(*Instances*)
	HMI:HMI_TemplateMachinePart;						//All HMI related variables
	Tmr_Empty:TON;										//Timer detection machine is empty*)
	Tmr_Initialisation:TON;								//Timer template*)
	Tmr_TestServoVelo:ton;
	Tmr_Wrn_NoSupply:ton;
	//Signal		>> outputs high / low. It can be used for any signal (that is not a sensor).
	SN_DscReadyToReceive:cntrl_InputHmiSts;					//Signal discharge ready to receive products
	//PB_Safe 		>> HMI safe button. This block automatically outputs low signal if the HMI loses connection for more than x-time
	PBsf_Example:utl_PB_HmiSafe;						//Safe pushbutton
	
	(*EXAMPLE how to init setpoint variables (normally you are not allowed to write these!) OR any variable of an instance
		use f2 >> select you setpoint type, for this I've chosen HMI_SP_Sensor >> insert with arguments >> this wil show up:
			HMI_SP_Sensor := (
				TMR_Muting:= , 
				TMR_DelayDetected:= , 
				TMR_DelayUndetected:= , 
				TMR_DelayErrorDetect:= , 
				TMR_DelayErrorUndetect:= );
		with this info you can init the setpoints of the cntrl_Sensor block like this:*)				
	
	//cntrl_Sensor	>> outputs: product detected / not detected. It can be used for any detection for example: airpressure, an object, etc.	
	//* If you init setpoints like this, then these values will only be used at first time download of the block. 
	// >> you will have to do a "plc" / "reset origin"
	PC_ProductInfeed:cntrl_Sensor(
		//fb_init
		Options:= eSensorConfig.InputNO)
		//Example how to preset setpoint variables
		:=(
			HMI:=(
				SP:=(
					TMR_DelayDetected:=T#100MS , 
					TMR_DelayUndetected:= T#101MS, 
					TMR_DelayErrorDetect:= T#2S1MS, 
					TMR_DelayErrorUndetect:= T#2S2MS)));	//Photocell product infeed position
	
	
	PC_PlanoBufferLL: cntrl_Sensor(
		Options:= eSensorConfig.Default);					//Photocell planobuffer low level 	
					
 
	//Valve			>> used to control cylinders with valves and reedcontacts
	Cyl_Example:cntrl_Valve
		(Options:= eValveConfig.Default);	

	//Motor			>> standard motor with forward/reverse + ana speed all direct IO
	Mtr_Example:cntrl_Motor(
		Options:= eMotorConfig.Default, 
		TmrDirectionChange:= T#500MS, 
		MinAllowedSpeed:= 25, 
		DAC_0PrctValue:= 0, 
		DAC_100PrctValue:= 0);
	
	//FreqDrive	ControlTechniques C300	>> Frequency drive motor, this one is controlled by ethercat
	Fdr_CtExample:cntrl_FDR_ControlTech(
		Options:= eFdrGeneric_Config.WithMaintSwitch, 
		UnitsToOutputFactor:= 30);

	//FreqDrive	Lenze I550 >> Frequency drive motor, this one is controlled by ethercat
	Fdr_LzExample:cntrl_FDR_Lenze(
		Options:= eFdrGeneric_Config.WithMaintSwitch, 
		UnitsToOutputFactor:= 30);

	//The interrol roller-drive BI can be used as frequency drive but also as a Cia402 positioning device >> for test configged as positioning device
	Srv_Interrol: cntrl_FDR_Interrol(
		Options:= eFdrGeneric_Config.ExternalRunStates, //this tells the base block to hand over control to the child block for the running-states 
		UnitsToOutputFactor:= 1);

	//Servo			>> Beckhoff servo drive
	Srv_Example:cntrl_Servo(
		TMR_PowerSave:=T#30S,			//time before entering powersave mode 0=disabled (if no command is given then power down after this time @ any command is reset timer) !It takes some time to awake the servo
		EnableSoftLimits:=FALSE,		//enable software limits (with button manual disable hw-limits, the parameter in the nc-task is set to 0, we need to know if it should be reenabled afterwards
		InputNrHomingSensor:=-1,			//input nr for the sensor in "axis_ref_Extended.I_DigitalInputs" -1 == disabled
		InputNrHwLimitNeg:=-1,			//input nr for the sensor in "axis_ref_Extended.I_DigitalInputs" -1 == disabled
		InputNrHwLimitPos:=4,			//input nr for the sensor in "axis_ref_Extended.I_DigitalInputs" -1 == disabled
		JogMinusOffHomeSensor:=FALSE,	//"jog-"  when moving off homing sensor (if false then jog+ is used) in homing function
		HomingsensorIs_NC:=FALSE,		//the homing sensor is of type normally closed (note limitswitches are always normally closed)
		TmrErr_JogOffHomeSensor:=T#3S,	//time to try and jog off homing sensor t#0S = disable
	
		HomeTorqueSpeed:=0,						//Speed to use for homing in torque mode
		HomingMode:= eSrvHomingModes.Direct,	//homing mode to use >> Default, Direct, Set, Reset, TorquePositiveDirection, TorqueNegativeDirection
		CouplingSyncPosFirst:=FALSE,			//at couple command, sync the position first to the master axis
		SPD_CouplingSyncSpeed:=0,				//speed to use when syncing position for coupling
		DST_CouplingSyncMaxDiff:=0,				//max difference allowed when sync couling >> otherwise error
		//MAKE SURE VALUE IS CORRECT (set to 0 to use nc-task configured dynamics)
		DEC_EmergencyError:=5000,				//deceleration ramp to use for emergency/error situation <= 0 means use default ramp
		//SET LOWER!!! >> jog=50, velo=250
		SPD_JOG_Max:=5000,						//max allowed allowed jog speed (also used to jog of homing sensor during homing)
		SPD_AbsModVel_MaxMan:=5000				//max allowed speed in manual absolute,velocity, modulo mode	
		);
	//Ganty			>> Gantry controlled with 2 beckhoff servo's connected to the same drive-belt
	Gantry_Example:cntrl_SingleBeltGantry(
			IsHomingUp:= TRUE, 
			IsHomingRight:= TRUE, 
			TMR_DelayPowerSave:= T#1M , 
			SPD_MaxJog:= 50, 
			SPD_MaxMove:= 150);
	
	//Robot			>>customized library robot block
	Rbt_Unloading: cntrl_RbtFanucUnloadingRobot();
			
	//VacuumGenerator	>>	Vacuumgenerator with blowoff controlled by IO
	Vcg_Suckers : cntrl_VacuumGenerator(
		//fb_init
		Options:= eVacuumGeneratorConfig.Default + eVacuumGeneratorConfig.DropVacAtVacErr)
		//interal vars
		:=(PS_VacuumOk:=(
			HMI:=(
				SP:=(
					TMR_DelayErrorDetect := T#2S,
					TMR_DelayErrorUnDetect := T#2S))));

	//Omron FH			>> Omron camera's controlled by an omron FH-controller over ethercat
	Cam_OmronFh: Cntrl_OmronFh;
	//Omron FH controlled by ethernet
	Cam_OmronFhEth: cntrl_OmronFhEth;
	Cam_OmronFhEthResult: utl_OmronFhEthResult_Template;
	Cam_OmronFhEthSimMessage:STRING := '1;65.9;85.4;-78.3;75;1;$R';

	//Omron smartcam	>> Omron smart camera's over ethernet / direct IO for trigger
	Cam_OmronSmartCam: Cntrl_OmronMicroScan(
		AlwaysConnected:= FALSE, 	//try to connect to camera even if no auto_k 
		JobNr:= 1, 					//default job nr to load if job load command is given (can be changed with property)
		UseIoTrigger:= FALSE);		//instead of trigger over ethernet, send trigger by real output
	

(*Inputs / Outputs*)
	//note> since there is a logged library input-block (cntrl_InputXXX) 
END_VAR

(*
	Update HMI variables
	Check if an error is active >> set Q_ProgStatus.Prog_Errror
*)
	HMI.M_Update(	I_OrgControl:= I_Organiser, 	//used for reset manuals/errors commands
					I_HMI_Parent := 0, 				//This is top level, no error propagation
					I_ERR:= HMI.ERR,				//The update function will check for error changes (signal to the hmi to update errors) + reset errors
					I_WRN:= HMI.WRN,				//The update function will check for warning changes (signal to the hmi to update errors)
					I_MAN:= HMI.MAN);				//The update function will reset manuals @ organiser request
			
(*	Simulation*)
	//if simulation active >> ..
	IF(Glbl.Sim_MyMachinePart) THEN A_Simulation();END_IF

(*	Exceptions & step-controller*)
	A_Exceptions();
		
(*	Step transitions*)
	//if not in exception >> execute step transitions
	IF (	NOT HM_ProgStatus.Prog_Exception)
	THEN 
		A_StepTransitions();
	END_IF
	
(*	Activations*)
	//Reset all outputs controlled by states
	A_ActivationsInit();
	//Activate outputs controlled by state
	A_ActivationsState();
	//Activate outputs not controlled by state + call all instances
	A_ActivationsAlways();
	
(*update organiser with scam status*)
	A_UpdateOrganiserProgstatus();

ACTION A_ActivationsAlways:
(*
	State undependant activations + instance calls
*)
//Internal flags
	//if running and product detected or supply might be supplying products > reset empty status
	IF (	I_Organiser.EnableDevices_K
			AND (	PC_ProductInfeed.Q_DetectedDebounced
					OR NOT I_STS_SUP_Empty))
	THEN
		HM_Empty := FALSE;
	END_IF

//Warnings/Statusses
	Q_STS_Empty := HM_Empty;
	HMI.STS.IsEmpty := HM_Empty; //can be used to indicate on the HMI this machinepart is empty
	Q_STS_RefillPlanos := NOT PC_PlanoBufferLL.Q_DetectedDebounced;
	HMI.WRN.PlanoBufferNeedsRefill := NOT PC_PlanoBufferLL.Q_DetectedDebounced;
	HMI.WRN.NotRdyRcv_Discharge := 	I_Organiser.EnableDevices_K
									AND NOT SN_DscReadyToReceive.Q;

	//if pulse 1s >> increase hmi test int until max reached which resets to 0
	IF(BknGlbl.Blink_P_1s)
	THEN
		HMI.STS.testInt := HMI.STS.testInt + 1; IF(HMI.STS.testInt > 5) THEN HMI.STS.testInt := 0; END_IF;
	END_IF

//Timers
	Tmr_Empty(	//IN:= ,
				PT:= T#30S );	
	
	Tmr_Initialisation(
		//IN:= ,
		PT:= T#3S);
		
	Tmr_TestServoVelo(	//IN:= , 
						PT:= T#5S);

//Instance calls
	//Safe button (protection against loss of communication with the HMI >> will set state to low)
	PBsf_Example();

	PC_ProductInfeed(
		I_HMI_Parent:= HMI,
		I_K_SimulationActive:= Glbl.Sim_MyMachinePart, 
		I_OrgControl := I_Organiser);
		//I_SimulateState:= ,
		//I_K_ErrNotState:= ,
	
	//Logged counter: example how we can count the debounced falling edges of a photocell
		IF(PC_ProductInfeed.Q_DetectedDebounced_RE) THEN 	PC_Example_Count.V := PC_Example_Count.V + 1; END_IF
	
	PC_PlanoBufferLL(
		I_HMI_Parent:= HMI,
		I_OrgControl:= I_Organiser,
		I_K_SimulationActive:= Glbl.Sim_MyMachinePart,
		I_SimulateState:= eSensorState.Detected, 
		I_ErrNotState:= eSensorState.None);
	
	SN_DscReadyToReceive(
		I_K_SimulationActive:= Glbl.Sim_MyMachinePart, 
		//I_K_SimulateOn:= 
		);
	
	Cyl_Example(
		I_HMI_Parent:= HMI,
		I_K_SimulationActive:= Glbl.Sim_MyMachinePart, 
		I_ES_OK:= I_K_ES_OK, 
		I_OrgControl:= I_Organiser,  
		//I_K_AutoIn:=,
		//I_K_AutoOut:=,
		);
		
	Vcg_Suckers(
		I_HMI_Parent:= HMI,
		I_K_SimulationActive:= Glbl.Sim_MyMachinePart,
		I_ES_OK:= I_K_ES_OK, 
		I_OrgControl:= I_Organiser, 
		//I_K_Auto_Vacuum:= , 
		//I_K_Auto_BlowOff:= , 
		);

	Mtr_Example(
		I_HMI_Parent:= HMI,
		I_K_SimulationActive:= Glbl.Sim_MyMachinePart, 
		I_ES_OK:= I_K_ES_OK, 
		I_OrgControl:= I_Organiser, 
		//I_K_Auto_Fwd:= , 
		//I_K_Auto_Rev:= , 
		I_Spd_AutoPrct:= -1, //>>use IO_SP.Spd_Default instead
	);
		
	Fdr_CtExample(
		I_HMI_Parent:= HMI,		
		I_K_SimulationActive:= Glbl.Sim_MyMachinePart, 
		I_ES_OK:= I_K_ES_OK, 
		I_OrgControl:= I_Organiser,  
		//I_K_Auto_Fwd:= ,
		//I_K_Auto_Rev:= , 
		//I_SPD_AutoPrct:= , 
		);
		
	Fdr_LzExample(
		I_HMI_Parent:= HMI, 
		I_K_SimulationActive:= Glbl.Sim_MyMachinePart, 
		I_ES_OK:= I_K_ES_OK, 
		I_OrgControl:= I_Organiser, 
		//I_K_RunFwd:= , 
		//I_K_RunRev:= , 
		//I_Speed:= 
		);
	
	
	//todo debug test
	Srv_Example.I_K_PosAbsolute R= HM_DebugServoRestart;
	Srv_Example(
		I_HMI_Parent:= HMI,
		I_PTR_MasterAxis:=0, 
		I_K_SimulationActive:= Glbl.Sim_MyMachinePart, 
		I_ES_OK:= I_K_ES_OK, 
		I_OrgControl:= I_Organiser, 
		//..several commands.. 
		I_CPF_CoupleFactor:= 1, 
		I_K_CoupleAxis:= FALSE, 
		I_K_UnCoupleAxis:= FALSE, 
		I_K_ExternalSetpoint:= FALSE); HM_DebugServoRestart := FALSE;
		
		(*log actual position / velocity. 
			*Constantly logging positions causes a lot of data for the logger!
			This is why in the servo block no position logging is done and you have to add it manually if you need it.
				>>decrease logging data volume by setting trigInterval and trigDeviation and add an elogGroup which is only activated when you need it
				>>Or only log at step transition
					IF(myStepCondition)
					THEN
						SRV_ExamplePos.V := TO_REAL(fbSrv_Example.P_STS_ActPosition);
						//>
						eMyStep:= blablabla;
					END_IF
		Done as below causes a lot of data
		*)
		Srv_Example_Velo.V := TO_REAL(Srv_Example.P_STS_ActVelocity); 
		
		(*Very specific example where the configuration is changed based on certain conditions>> for this example normally the man-speeds are only set in fb_init()*)
		//if in manual mode
		IF(I_Organiser.Manual_K AND FALSE)
		THEN
			//if servo is NOT coupled >> limit to lower value for safety
			IF(NOT Srv_Example.P_STS_IsCoupled) 
			THEN 
				Srv_Example.P_CFG_SPD_ABSMODVEL_MaxMan := 5;
				Srv_Example.P_CFG_SPD_JOG_MaxMan := 5;
			ELSE
				Srv_Example.P_CFG_SPD_ABSMODVEL_MaxMan := 500;
				Srv_Example.P_CFG_SPD_JOG_MaxMan := 100;
			END_IF
		END_IF
		
	Srv_Interrol(
		I_HMI_Parent:= HMI, 
		I_OrgControl:= I_Organiser, 
		I_K_SimulationActive:= Glbl.Sim_MyMachinePart, 
		I_ES_OK:= I_K_ES_OK, 
		I_K_Auto_Fwd:= FALSE, 		//not used in this example (can be used!) 
		I_K_Auto_Rev:= FALSE, 
		I_Speed:= -1,				// <0 = block will use internal setpoint value 
		//I_K_AbsPositioning:= , 	//only used command in this example
		//I_Position:= , 
		);
	
	Gantry_Example(
		I_HMI_Parent:= HMI,
		I_K_SimulationActive:= Glbl.Sim_MyMachinePart,
		I_ES_OK:= I_K_ES_OK, 
		I_OrgControl:= I_Organiser,
		//I_Auto_K_Homing:= , 
		//I_Auto_K_MoveToPos:= , 
		//I_Auto_POS_MoveToPos:= , 
		//I_Auto_SPD_MoveToPos:= 
	);
	
	Rbt_Unloading(
		I_HMI_Parent:= HMI, 
		I_OrgControl:= I_Organiser, 
		I_K_SimulationActive:= Glbl.Sim_MyMachinePart, 
		I_ES_OK:= I_K_ES_OK, 
		I_K_ProgramSelect:= , 
		I_SP_ProgramNr:= , 
		Q_K_ProgramSelect_OK=> );
	
	Cam_OmronSmartCam(
		I_HMI_Parent:= HMI,
		I_K_SimulationActive:= Glbl.Sim_MyMachinePart,
		I_OrgControl:= I_Organiser, 
		//I_K_Trigger:= , 
		//I_K_AutoCal:= , 
		//I_K_QuickFocus:= , 
		//I_K_LoadJob:= , 
		IO_DataReceive:= HM_CamReceivedData, 
		);
		//just for debugging, should be removed
		//data should normally be handled at the state transition when waiting for trigger ok
		IF(Cam_OmronSmartCam.Q_K_Trigger_Ok)
		THEN
			//note: this boikon library block will take care not to overflow the destination memory
			utl_Any_CopyWithOffset(
				I_Destination:= HMI.STS.OmronSmartCamLastResult, 
				I_Source:= HM_CamReceivedData, 
				I_WriteOffset:= 0);
		END_IF
		
	Cam_OmronFh(
		I_HMI_Parent:= HMI,
		I_K_SimulationActive:= Glbl.Sim_MyMachinePart,
		I_OrgControl:= I_Organiser,
		//I_K_Trigger:= , 
		//I_K_TriggerNextResult:= , 
		//I_K_ChangeGroup:= , 
		//I_K_LoadScene:= , 
		//I_SceneToLoad:= , 
		);
	
	(*Simple example of handling data received by controller. 
	I recommend doing this in the step transition and directly connect it to the desired location and using return value of the function instead of doing it here
	the disadvantage of doing it like this that everything inside the block is executed continiously and hogs the processor.
	Recommended way @ step transitions: 
		IF(utl_OmronCameraResult(..,..,myBuffer)) 
		THEN 
			//>>
			eS:=xxx.CamResultOK;
		ELSE
			//>>
			eS:= xxx.CamResultNOK;
		..
	*) 

	Cam_OmronFhEth(
		I_HMI_Parent:= HMI, 
		I_K_SimulationActive:= Glbl.Sim_MyMachinePart,
		I_SimulationTrigResult:= Cam_OmronFhEthSimMessage,
		I_OrgControl:= I_Organiser, 
		I_ReceiveBuffer:= HM_CamOmronFhEthReceivedData, 
		I_K_LoadScene:= ,
		I_K_UpdateStatus:= , 
		//I_K_Trigger:= 
			);
			
		//block that will resolve results from camera measurement output
		Cam_OmronFhEthResult(
			I_K_TrigOk:= Cam_OmronFhEth.Q_K_TriggerOk,
			I_DataUsedSize:= Cam_OmronFhEth.Q_STS_TriggerNrBytesReceived, 
			I_Data:= HM_CamOmronFhEthReceivedData);
END_ACTION

ACTION A_ActivationsInit:
(*	
	Initialisation of state dependant activations
*)
HM_ProgStatus.Prog_Rest := FALSE;
Q_SN_SUP_Request := FALSE;
PC_ProductInfeed.I_ErrNotState := eSensorState.None;
Mtr_Example.I_K_Auto_Fwd := FALSE;
Mtr_Example.I_K_Auto_Rev := FALSE;
Fdr_CtExample.I_K_Auto_Fwd := FALSE;
Fdr_CtExample.I_K_Auto_Rev := FALSE;
Fdr_LzExample.I_K_Auto_Fwd := FALSE;
Fdr_LzExample.I_K_Auto_Rev := FALSE;
Cyl_Example.I_K_AutoIn := FALSE; 
Cyl_Example.I_K_AutoOut := FALSE;
Vcg_Suckers.I_K_Auto_BlowOff :=FALSE;
Vcg_Suckers.I_K_Auto_Vacuum :=FALSE;
Srv_Example.I_K_Homing:= FALSE;
Srv_Example.I_K_PosAbsolute:= FALSE;
Srv_Example.I_K_Velocity := FALSE;
Srv_Interrol.I_K_AbsPositioning := FALSE;
Cam_OmronFh.I_K_Trigger := FALSE;
Cam_OmronFh.I_K_TriggerNextResult := FALSE;
Cam_OmronFh.I_K_ChangeGroup:= FALSE;
Cam_OmronFh.I_K_LoadScene:= FALSE;
Cam_OmronFhEth.I_K_Trigger:= FALSE;
Cam_OmronSmartCam.I_K_AutoCal := FALSE;
Cam_OmronSmartCam.I_K_LoadJob := FALSE;
Cam_OmronSmartCam.I_K_QuickFocus := FALSE;
Cam_OmronSmartCam.I_K_Trigger := FALSE;
Rbt_Unloading.I_K_DropBasket := FALSE;


Tmr_Empty.IN := FALSE;
Tmr_TestServoVelo.IN := FALSE;
Tmr_Initialisation.IN := FALSE;
Tmr_Wrn_NoSupply.IN := FALSE;

HM_DebugMultiStep_ResetInActivations := false;
END_ACTION

ACTION A_ActivationsState:
(*
	State dependant activations
*)
CASE State.eS OF
	eTMP.TotalReset:
		;
	
	eTMP.InitCyl:
		Cyl_Example.I_K_AutoIn:= TRUE; 
	
		(*Warnings/Errors*)
			//a sensor error can be triggered by activating the I_K_ErrNot.... input >> uses internally a timer
			//usually we want the machine to be empty in the init phase so setting error here if it is not
			PC_ProductInfeed.I_ErrNotState := eSensorState.Undetected; 
			//or an error can also be set directly
			//IF( [some condition] ) then IO_ERR.PC_ProductPassedStopper.NotLow := true; END_IF  !!!Errors must be a set! 
	
	eTMP.InitSrv:
		Cyl_Example.I_K_AutoIn:= TRUE; 
		Mtr_Example.I_K_Auto_Fwd:= TRUE;
		Srv_Example.I_K_Homing:= TRUE;
		Tmr_Initialisation.IN:= Mtr_Example.P_STS_Running;
	
		(*Warnings/Errors*)
			//S= >> SET!!! , all errors have to be set. In tc3 we can now use S= instead of "IF(..)THEN err:=true; end_if"
			HMI.ERR.InitNotEmpty S= PC_ProductInfeed.Q_DetectedDebounced;  	//detection machine is not empty during init
			PC_ProductInfeed.I_ErrNotState := eSensorState.Undetected;			//it is nice to also trigger this error, especially if there are multiple sensors. This at a faulty sensor the operator knows which sensor causes the problem
	
	eTMP.InitCamQuickFocus:
		Cyl_Example.I_K_AutoIn:= TRUE; 
		Cam_OmronSmartCam.I_K_QuickFocus:= TRUE;
	
	eTMP.InitCamLoadJob:
		Cyl_Example.I_K_AutoIn:= TRUE; 
		Cam_OmronFh.I_K_LoadScene:= TRUE;
		Cam_OmronFh.I_SceneToLoad:= 2;
		Cam_OmronSmartCam.I_K_LoadJob:= TRUE;
		Cam_OmronSmartCam.P_SP_JobToLoad:= 1; //note: these kind of variables can also be set @RE step (>>when stepping from previous step to here)			(*Internals*)
			
	eTMP.Rest:
		HM_ProgStatus.Prog_Rest:= TRUE;
		Q_SN_SUP_Request:= TRUE;
		Cyl_Example.I_K_AutoIn:= TRUE; 
		
		(*Warnings/Errors*)
			//just an example, no need to add this specific warning. The camera itself generates an error if it fails to connect
			HMI.WRN.CameraNotReady:= 	I_Organiser.EnableDevices_K
										AND NOT Cam_OmronSmartCam.Q_STS_Ready;  
			
			//if the supply is running >> the photocell should get high after x-time, set error detection of the pc
			IF(	I_SN_SUP_Request_OK
				AND NOT I_STS_SUP_Empty
				AND I_Organiser.EnableDevices_K)
			THEN
				PC_ProductInfeed.I_ErrNotState:= eSensorState.Detected; 
			END_IF

	eTMP.SrvPosStart:
		Cyl_Example.I_K_AutoIn:= TRUE; 
		Srv_Example.I_K_PosAbsolute:= TRUE;
		//there are multiple ways of setting a speed, this way per step the speed can be changed but it can also set fixed at the servo block
		//also note how for the gripper, settings are applied at the step change >>better way if during the step the settings do not have to change
		Srv_Example.I_SP_Speed:= 50;
		Srv_Interrol.I_K_AbsPositioning := TRUE; 
		
	eTMP.SrvPosStartInterl:
		Cyl_Example.I_K_AutoIn:= TRUE;
		Rbt_Unloading.I_K_DropBasket := true;
		
		(*Warnings/Errors*)
			PC_ProductInfeed.I_ErrNotState:= eSensorState.UnDetected; 

	eTMP.SrvPosEnd:
		Cyl_Example.I_K_AutoIn:= TRUE;
		Srv_Example.I_K_PosAbsolute:= TRUE;
		Srv_Example.I_SP_Speed:= 50; //there are multiple ways of setting a speed, this way per step the speed can be changed but it can also set fixed at the servo block
		Srv_Interrol.I_K_AbsPositioning := TRUE;
		
	eTMP.SrvPosEndIntrl:
		Cyl_Example.I_K_AutoIn:= TRUE;
		
	eTMP.CylOut:
		Cyl_Example.I_K_AutoOut:= TRUE;
		Vcg_Suckers.I_K_Auto_Vacuum:=TRUE;
		
	eTMP.CylIn:
		Cyl_Example.I_K_AutoIn:= TRUE;
		Vcg_Suckers.I_K_Auto_BlowOff:=TRUE;	
		
	eTMP.MtrStartFwd:
		Cyl_Example.I_K_AutoIn:= TRUE;	
		Mtr_Example.I_K_Auto_Fwd:= TRUE;

		//fdr's speed = block input
		Fdr_CtExample.I_K_Auto_Fwd:= TRUE;
		Fdr_CtExample.I_Speed:= -1; //<0 means use HMI.SP.Speed
		Fdr_LzExample.I_K_Auto_Fwd:= TRUE;
		Fdr_LzExample.I_Speed := 50;
		
	eTMP.MtrStop:
		Cyl_Example.I_K_AutoIn:= TRUE;
	
	eTMP.MtrStartRev:
		Cyl_Example.I_K_AutoIn:= TRUE;	
		Mtr_Example.I_K_Auto_Rev:= TRUE;

		//fdr's speed = HMI.SP
		Fdr_CtExample.I_K_Auto_Rev:= TRUE;
		Fdr_CtExample.I_Speed:= 75; //<0 means use HMI.SP.Speed
		Fdr_LzExample.I_K_Auto_Rev:= TRUE;
		Fdr_LzExample.I_Speed := -1; //<0 means use HMI.SP.Speed

	eTMP.CamReady:
		Cyl_Example.I_K_AutoIn:= TRUE;			
	
	eTMP.CamTrig:
		Cyl_Example.I_K_AutoIn:= TRUE;
		Cam_OmronFh.I_K_Trigger:= TRUE;
		Cam_OmronFhEth.I_K_Trigger:= TRUE;
		Cam_OmronSmartCam.I_K_Trigger:= TRUE;	
		
(*
	S_Example:
		//Comm signals
		//Timers
		//Internals
		//Controls
		//Warnings
		//Errors
*)

END_CASE
END_ACTION

ACTION A_Exceptions:
(* State transition controller
	Handles multistep + step hold + statusses for hmi + logging*) 
		//>>must be before all method calls, since the input arguments are used
	State(I_OrgControl := I_Organiser);

(*Exceptions
	Here exeptions are handled.
	*most basic version:
		Rest U_0 := Q_ProgStatus.Prog_Exception:=false
			the main program is executed
	
		Rest >> Error := Q_ProgStatus.Prog_Exception:=true
		1)	@ any error >> exception state (U1_0)
			this will freeze the main program states
		2)	if the organiser is back in an automatic state and there are no errors
			it will step to U1_2 and from there to the idle state U_0
			*TODO TEMPLATE >> if needed, do actions on this transition (rarely used)
				But you could for example at a specific error force the main program to a recovery step
			
			
		Rest >> Totalreset := Q_ProgStatus.Prog_Exception:=true
		1)	@ organiser total reset command >> exception total reset (U1_1)
		
		2)	@ NOT organiser total reset command >> 
				>> now bits that need to be reset @ total reset are reset
				TODO Template >> add bits which needs to be reset
				>> the main program is reset to the first step (usually named: TotalReset)
				>>back to rest (U_0)

	**this described the basic version which can be used in 99% of the cases,
	you can adapt it to your needs. 
*)

CASE eE OF
	//rest
	U_0:
		
		//if program in error >> to error state
		IF(	HM_ProgStatus.Prog_Error
			AND NOT I_Organiser.TotalReset_K)
		THEN
			//>>
			eE := U1_0;
		//else if total reset command >> to total reset state
		ELSIF(	I_Organiser.TotalReset_K)
		THEN
			//>>
			eE := U1_1;
		END_IF

	//error
	U1_0:
		//if total reset command >> to total reset state
		IF(	I_Organiser.TotalReset_K)
		THEN
			//>>
			eE := U1_1;
			
		//else if no error active and organiser back in an automatic state
		ELSIF(	NOT HM_ProgStatus.Prog_Error
				AND I_Organiser.EnableDevices_K)
		THEN
			//>>
			eE := U1_2;
		END_IF

	//Total Reset
	U1_1:
 		//if total reset command dropped >> Reset program data and to unfreeze state
		IF(	NOT I_Organiser.TotalReset_K)
		THEN
			//Total reset main program
			State.M_Step(
				I_NewStep:= eTMP.TotalReset,
				I_StepCanBeHeld:= TRUE);
			
			//disable multistepping for 1 round
			{warning disable C0139}
			State.P_IsMultiStepRequired;

			//Reset main program flags
			HM_Empty:=FALSE;
			//only done as example/testing, should be removed
			HMI.ERR.ExampleAddPrioForHmiError := TRUE;
			
			//>>
			eE := U_0;
		END_IF
		
	//Unfreeze
	U1_2:
		//>>
		eE := U_0;

	ELSE
		eE := U_0;
END_CASE

//Detection program in exception
HM_ProgStatus.Prog_Exception := (eE > U_0);
END_ACTION

ACTION A_Simulation:
(*
	Code that only needs to be executed if simulation is active (this action is only called if sim is active)

	Notes:	
	-Cntrl_Servo/motor/valve already simulate their state correctly themselves, cntrl_StateSensor must be told which state to simulate >> example below
		Of course you could also add timers / other conditions (servo pos?!) for states
	
	-you can use ( Tmr_StateTime.PT > T# xxx) to start simulating things after the state has been active for a certain time
*)

//Initialise activations, which are controlled by the simulation steps
SN_DscReadyToReceive.I_K_SimulateOn := FALSE;
PC_ProductInfeed.I_SimulateState := eSensorState.Undetected;

(*Step activations*)
CASE State.eS OF
	eTMP.TotalReset:
	;

	eTMP.InitCyl:
	;
	
	eTMP.InitSrv:
	;

	eTMP.Rest:
		PC_ProductInfeed.P_BypassErrDetectionTime := State.P_StepTime + T#100MS; 
		
		//If delay time elapsed >> simulate sensor + discharge request
		IF(State.P_StepTime > T#1S) 
		THEN
			SN_DscReadyToReceive.I_K_SimulateOn := TRUE; 
			PC_ProductInfeed.I_SimulateState := eSensorState.Detected;
		END_IF
		
	eTMP.SrvPosStart:
	;
		
	eTMP.SrvPosStartInterl:
	;
END_CASE	

//feedback request to input
I_SN_SUP_Request_OK := Q_SN_SUP_Request;
END_ACTION

ACTION A_StepTransitions:
(*In this section all state transitions are made

	-no activations are done here (do this in A_Activations)
	-The transition to a new step is the ideal location to do rising edge settings
		IF(myCondition) THEN
			HM_CNT_Example := HM_CNT_EXAMPLE + 1; //example to count something
			fbSrv_Example.I_POS_Auto_Absolute := myNewPosition + someCalculated offset; //example to calculate endpoint for a servo
			//Note: you could set the servo speed here as well, but then you can't change the speed anymore during the movement
				probably (dependant on your situation) better to do it in activations.
			//>>
			step to next step
		END_IF

*)

(*Main program steps*)

//if stepping not locked, by steplock mode >> can be toggled in HMI to lock certain steps for commissioning/debugging
IF( NOT State.Q_K_LockSteps)
THEN
//Repeat until conditions to step to next state are false OR looped already twice (normally programs don't loop multiple times!)
REPEAT 
	CASE State.eS OF
		eTMP.TotalReset:
			//if initialise command from the organiser >> start initialisation
			IF ( I_Organiser.Init_K)
			THEN
				//>>
				State.M_Step(
					I_NewStep:= eTMP.InitCyl,
					//Optional: argument to log extra info for this step transition
					I_NewStepLogInfo:= CONCAT('TotalReset:', SYSTEMTIME_TO_STRING(BknGlbl.LocalSystemTime)),
					//>>@ true & HMI-stepmode is activated, then the next state will be locked until you press the button release step on the HMI (used for debugging / commissioning
					//!Do not enable for states in which things are cooking: (heater enabled / motor running / etc) or at least consider carefully potential dangers.
					I_StepCanBeHeld:= TRUE,
					//Optional: >> the repeat around this CASE-statement will NOT execute, the next step will take at least 1 cycle == activations for that step are executed 	
					I_BlockMultiStep:=TRUE); 
			END_IF

		
		eTMP.InitCyl:
			//if cylinder initialised and no products in the machine >> InitSrv
			IF( Cyl_Example.Q_STS_In
				AND NOT PC_ProductInfeed.Q_DetectedDebounced) //note: >> set error detection in activations!
			THEN
				//>>
				State.M_Step(
					I_NewStep:= eTMP.InitSrv,
					I_StepCanBeHeld:= TRUE);
			END_IF
			
		eTMP.InitSrv:
			//if servos homed and minimal time elapsed >> next state
			IF( Srv_Example.Q_K_HomingOk
				AND Tmr_Initialisation.Q) 
			THEN
				//>>
				State.M_Step(
					I_NewStep:= eTMP.InitCamQuickFocus,
					I_StepCanBeHeld:= TRUE);
			END_IF
			
		eTMP.InitCamQuickFocus:
			//if camera ready / quickfocus done >>..
			IF(	Cam_OmronFh.Q_STS_Ready
				AND Cam_OmronSmartCam.Q_K_AutoOrQuickCal_Ok)
			THEN
				//>>
				State.M_Step(
					I_NewStep:= eTMP.InitCamLoadJob,
					I_StepCanBeHeld:= TRUE);
			END_IF
			
		eTMP.InitCamLoadJob:
			//if camera's loaded jobs >. ..
			IF(	Cam_OmronFh.Q_SN_LoadScene_OK
				AND Cam_OmronSmartCam.Q_K_LoadJob_Ok)
			THEN
				//>>
				State.M_Step(
					I_NewStep:= eTMP.Rest,
					I_StepCanBeHeld:= TRUE);
			END_IF

		eTMP.Rest: 
			//if in automatic mode and supply delivered product and interlockings ok
			//>>SrvPosStart
			IF( I_Organiser.Auto_K
				AND NOT HM_Empty					//machine is not empty (inclusive supply)
				AND I_SN_SUP_Request_OK				//supply delivered product
				AND SN_DscReadyToReceive.Q 			//discharge is requesting products
 				AND PC_ProductInfeed.Q_DetectedDebounced 	//expected the sensor to be high >> activate error monitoring in activations

				//interlocking >> check blocks returned to rest/ready state
				AND Cam_OmronFh.Q_STS_Ready
				AND Cam_OmronFhEth.Q_STS_Ready
				AND Cam_OmronSmartCam.Q_STS_Ready
				AND Cyl_Example.Q_STS_In
				AND NOT Vcg_Suckers.Q_K_BlowOffOK 	
				AND NOT Vcg_Suckers.Q_K_VacuumOK
				AND NOT Srv_Example.Q_K_PosAbsoluteOk
				AND NOT Srv_Interrol.Q_STS_TargetReached)
			THEN
				//setting positions on step change, you could also constantly write these positions constantly in activations
				Srv_Example.I_SP_Position:= HMI.SP.POS_SrvBegin;
				Srv_Interrol.I_Position:= HMI.SP.POS_SrvBegin;
				
				//example on how to avoid concat(concat(concat(concat......)))))
				//NOTE: it is not the most performant because of all the fancy c#-linq-like stuff but it is the simplest and faster than concat
				// 		really fast is using utl_Any_CopyWithOffset directly (the databuilder is a wrapper around that function)
				DataBuilder.
					//assign databuffer
					M_SetTarget(HM_InfoString).
					//add a string that is not a variable otherwise use: M_WithData(HM_MyStringVar)
					M_WithStringLiteral('Last cycle time:').
					M_WithStringLiteral(TO_STRING(TO_REAL(BknGlbl.SystemTimeInTicks - HM_LastTicksStateRest)/10000000)).
					M_WithStringLiteral('s Servos target pos:').
					M_WithStringLiteral(TO_STRING(HMI.SP.POS_SrvBegin)); 
					
				//>>
				State.M_Step(
					I_NewStep:= eTMP.SrvPosStart,
					//just an example what you can do (add state info for logging purposes), this argument is optional
					I_NewStepLogInfo:= HM_InfoString,
					I_StepCanBeHeld:= FALSE);
				
				HM_LastTicksStateRest := BknGlbl.SystemTimeInTicks;	
			//if in semi-automode and the operator choose a special action >> do requested action
			ELSIF( 	I_Organiser.SemiAuto_K
					AND TRUE) //insert HMI.STS.TB_RequestSpecialAction
			THEN
				
				//>>
				State.M_Step(
					I_NewStep:= eTMP.SemiAutoStart,
					I_StepCanBeHeld:= TRUE);
					
				HM_LastTicksStateRest := BknGlbl.SystemTimeInTicks;
			END_IF

		eTMP.SrvPosStart:
			//if servo's reached commanded position
			IF( Srv_Example.Q_K_PosAbsoluteOk
				AND Srv_Interrol.Q_STS_TargetReached
				//interl. make sure not still high from previous action
				AND NOT Rbt_Unloading.Q_K_DropBasket_OK)
			THEN
				//>>
				State.M_Step(
					I_NewStep:= eTMP.SrvPosStartInterl,
					I_StepCanBeHeld:= TRUE); //enabling step lock, so we can see at the machine how the servo is positioned if done 
			END_IF
		
		eTMP.SrvPosStartInterl:
			//if robot done and interlockings with servo/supply done
			//>>SrvPosEnd
			IF( 	Rbt_Unloading.Q_K_DropBasket_OK
					AND NOT PC_ProductInfeed.Q_DetectedDebounced			//let's also check the sensor dropped again >> make sure to trigger error detection in activations
					AND NOT I_SN_SUP_Request_OK					//product was handled, check if supply acknowledges
					//interl. next step a command is given so we need to interlock here
					AND NOT Srv_Example.Q_K_PosAbsoluteOk
					AND NOT Srv_Interrol.Q_STS_TargetReached)		
			THEN
				//again setting position on step change, you could also constantly write these positions constantly in activations
				Srv_Example.I_SP_Position := HMI.SP.POS_SrvEnd;
				Srv_Interrol.I_Position:= HMI.SP.POS_SrvEnd;
				
				//>>
				State.M_Step(
					I_NewStep:= eTMP.SrvPosEnd,
					I_StepCanBeHeld:= FALSE);
			END_IF
			
		eTMP.SrvPosEnd:
			//if servo reached end position
			//>>SrvPosEndIntrl
			IF(	Srv_Example.Q_K_PosAbsoluteOk
				AND Srv_Interrol.Q_STS_TargetReached)
			THEN
				//>>
				State.M_Step(
					I_NewStep:= eTMP.SrvPosEndIntrl,
					I_StepCanBeHeld:= TRUE); //enabling step lock, so we can see at the machine how the servo is positioned if done	
			END_IF
			
		eTMP.SrvPosEndIntrl:
			//if servo interlocking done >> CylOut
			IF(	NOT Srv_Example.Q_K_PosAbsoluteOk
				AND NOT Srv_Interrol.Q_STS_TargetReached)
			THEN
				//>>
				State.M_Step(
					I_NewStep:= eTMP.CylOut,
					I_StepCanBeHeld:= FALSE);				
			END_IF
			
		eTMP.CylOut:
			//if cylinder is out and product grabbed with vacuum >> CylIn 
			IF( Cyl_Example.Q_STS_Out
				AND Vcg_Suckers.Q_K_VacuumOK)
			THEN
				//>>
				State.M_Step(
					I_NewStep:= eTMP.CylIn,
					I_StepCanBeHeld:= TRUE);
			END_IF

		eTMP.CylIn:
			//if cylinder is in and actions done >> MtrStartFwd
			IF( Cyl_Example.Q_STS_In
				AND NOT Vcg_Suckers.Q_K_VacuumOK
				AND Vcg_Suckers.Q_K_BlowOffOK
				//interlocks !note added extra interlocks just for unittesting you don't need to do this with these blocks
				AND NOT Mtr_Example.P_STS_Running
				AND Fdr_CtExample.Q_STS_Stopped
				AND NOT Fdr_CtExample.Q_STS_TargetReached
				AND Fdr_LzExample.Q_STS_Stopped
				AND NOT Fdr_LzExample.Q_STS_TargetReached)
			THEN
				//>>
				State.M_Step(
					I_NewStep:= eTMP.MtrStartFwd,
					I_StepCanBeHeld:= FALSE);
			END_IF	

		eTMP.MtrStartFwd:
			//if all motors started
			//>>MtrStop
			IF( Mtr_Example.P_STS_Running
				AND Fdr_CtExample.Q_STS_TargetReached
				AND Fdr_LzExample.Q_STS_TargetReached
				//interl.
				AND NOT Vcg_Suckers.Q_K_BlowOffOK)
			THEN
				//init flag
				HM_MtrRevDone:= FALSE;
				//>>
				State.M_Step(
					I_NewStep:= eTMP.MtrStop,
					I_StepCanBeHeld:= TRUE);
			END_IF
			
		eTmp.MtrStop:
			//if all motors stopped
			//>>MtrStartRev/CamReady
			IF(	NOT Mtr_Example.P_STS_Running
				AND Fdr_CtExample.Q_STS_Stopped
				AND NOT Fdr_CtExample.Q_STS_TargetReached 
				AND Fdr_LzExample.Q_STS_Stopped
				AND NOT Fdr_LzExample.Q_STS_TargetReached)
			THEN
				//if motors not ran reverse yet 
				//>>MtrStartRev
				IF(NOT HM_MtrRevDone)
				THEN
					//>>
					State.M_Step(
						I_NewStep:= eTMP.MtrStartRev,
						I_StepCanBeHeld:= FALSE);
				//else motor cycle done
				//CamReady
				ELSE				
					//>>
					State.M_Step(
						I_NewStep:= eTMP.CamReady,
						I_StepCanBeHeld:= TRUE);
				END_IF
			END_IF

		eTMP.MtrStartRev:
			//if all motors started
			//>>MtrStop   NOTE: this is a bit ugly.. neater to just program the extra step
			IF( Mtr_Example.P_STS_Running
				AND Fdr_CtExample.Q_STS_TargetReached
				AND Fdr_LzExample.Q_STS_TargetReached)
			THEN
				//set flag
				HM_MtrRevDone:=TRUE;
				
				//>>
				State.M_Step(
					I_NewStep:= eTMP.MtrStop,
					I_StepCanBeHeld:= TRUE);
			END_IF
			
		eTmp.CamReady:
			//if camera's ready   NOTE: this extra step is not really needed conditions could have been added from rest>>xxx
			//>>CamTrig
			IF(	Cam_OmronFh.Q_STS_Ready
				AND Cam_OmronFhEth.Q_STS_Ready
				AND Cam_OmronSmartCam.Q_STS_Ready
				//interlockings
				AND NOT Cam_OmronFh.Q_SN_Trigger_OK
				AND NOT Cam_OmronFh.Q_SN_Trigger_NOK
				AND NOT Cam_OmronFhEth.Q_K_TriggerOk
				AND NOT Cam_OmronSmartCam.Q_K_Trigger_Ok
				AND NOT Cam_OmronSmartCam.Q_K_Trigger_Nok)
			THEN
				//>>
				State.M_Step(
					I_NewStep:= eTMP.CamTrig,
					I_StepCanBeHeld:= TRUE);
			END_IF

		eTmp.CamTrig:
			//if camera's done triggering
			//>>CamTrig
			IF(	(	Cam_OmronFh.Q_SN_Trigger_OK
					OR Cam_OmronFh.Q_SN_Trigger_NOK)
				AND 	Cam_OmronFhEth.Q_K_TriggerOk
				AND (	Cam_OmronSmartCam.Q_K_Trigger_Ok
						OR Cam_OmronSmartCam.Q_K_Trigger_NOk))
			THEN
				HM_DebugMultiStep_ResetInActivations := TRUE; //used for testing multistepping
				
				//>>
				State.M_Step(
					I_NewStep:= eTMP.MultiStepTest2,
					I_StepCanBeHeld:= TRUE);
			END_IF			
			

		//Example what multistepping does
		//if condition for next state is true then fall through to the next step in the same cycle
		//this prevents a device possibly being activated for only 1 cycle when falling through a rest step
		//>>in this example if the program gets to activations, this state will never be high (already fallen through when we get there).
		eTMP.MultiStepTest2:
			//if multistepping is working, this step will not be high for 1 cycle. It will fall through
			IF(TRUE)
			THEN
				//>>
				State.M_Step(
					I_NewStep:= eTMP.MultiStepTest3,
					I_StepCanBeHeld:= FALSE);				
			END_IF

		//In this step multistepping is tested if it stops after counting more than 1 back step.			
		eTMP.MultiStepTest3:
			//if testing multistepping hang >> try to hang multistepping
			IF(HM_DebugMultiStep_ResetInActivations)
			THEN
				//>>
				State.M_Step(
					I_NewStep:= eTMP.MultiStepTest2,
					I_StepCanBeHeld:= FALSE);				
			//else done testing multistepping >> back to rest
			ELSE

				//>>
				State.M_Step(
					I_NewStep:= eTMP.Rest,
					I_StepCanBeHeld:= FALSE);	
			END_IF		

		eTMP.SemiAutoStart:
			IF( State.P_StepTime > T#2S)
			THEN
				//>>
				State.M_Step(
					I_NewStep:= eTMP.SemiAutoStop,
					I_StepCanBeHeld:= TRUE);
					
			//example how to abort operation before anything happened					
			ELSIF(NOT I_Organiser.SemiAuto_K)
			THEN
				//>>
				State.M_Step(
					I_NewStep:= eTMP.Rest,
					I_StepCanBeHeld:= TRUE);
			END_IF
			
		eTMP.SemiAutoStop:
		//note: this will cause a deadlock, I'm doing it on purpose here to test things.
		//*the program should always be able to return to a rest-step before you add another Semi-/Auto_K condition
			IF( I_Organiser.SemiAuto_K
				AND State.P_StepTime > T#2S)  
			THEN
				//>>
				State.M_Step(
					I_NewStep:= eTMP.Rest,
					I_StepCanBeHeld:= TRUE);
			END_IF
			
	//unkown state, should never happen. Best to not do an autorecovery, just let it hang			
	ELSE
		utl_SystemMessageWithLogging(I_Message:='prog error step missing');
	END_CASE  

//until flag to multistep is false 
UNTIL(NOT State.P_IsMultiStepRequired)
END_REPEAT
END_IF
END_ACTION

ACTION A_UpdateOrganiserProgstatus:
//machinepart in exception > done in A_Exceptions
//HM_ProgStatus.Prog_Exception

//machinepart in rest state > done in A_ActivationsState
//HM_ProgStatus.Prog_Rest

HM_ProgStatus.Prog_Error :=	//emergencystop not ok
							NOT I_K_ES_OK
							//error active in this block or one of the local children (cntrl_xxxx for example)
							OR HMI.P_STS_InError;

//production stopped by external factor >> for OEE performance tracking / lamp signal column 
HM_ProgStatus.Prog_ExternallyBlocked := NOT SN_DscReadyToReceive.Q;

//machinepart needs attention >> for lamp signal column
HM_ProgStatus.Prog_Attention := PC_PlanoBufferLL.Q_DetectedDebounced;

//call organiser update method
I_Organiser.M_UpdateProgStatus(HM_ProgStatus);
END_ACTION

END_FUNCTION_BLOCK

// ---- DevelopmentPlayground/UnitTesting/Vis_Test.TcVIS
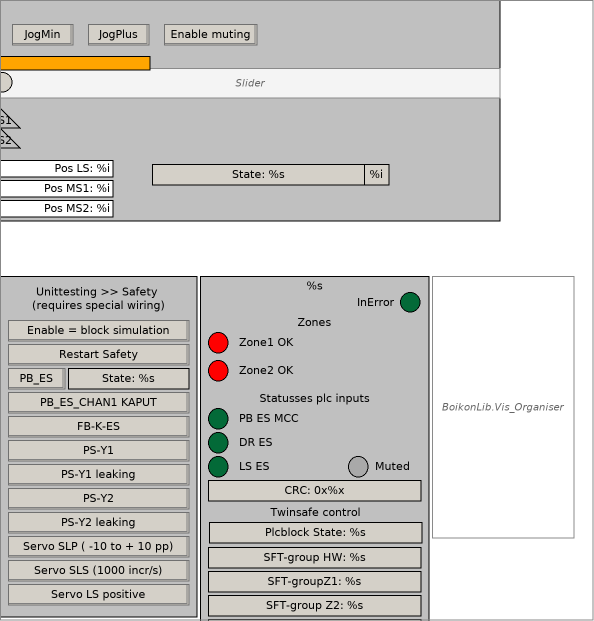
VISUALIZATION Vis_Test  // 594x621
    Rectangle (0,0 500x221)
    Slider (0,68 500x30), variable: UnitTesting.Sft_LS_PosBox, scale 0..485
    Rectangle (0,56 150x14)
        p3560616238: UnitTesting.Sft_LS_PosBox + 0
    Polyline (-20,128) (0,108) (20,128) (-20,128), "MS1", colour toggle: UnitTesting.Qsf_LS_Muting1
        p3560616238: UnitTesting.Sft_LS_PosMS1 + 0
    Polyline (-20,148) (0,128) (20,148) (-20,148), "MS2", colour toggle: UnitTesting.Qsf_LS_Muting2
        p3560616238: UnitTesting.Sft_LS_PosMS2 + 0
    Line (0,20) (0,152), colour toggle: UnitTesting.Qsf_LS_OSSD
        p3560616238: UnitTesting.Sft_LS_PosLS
    Rectangle (0,160 113x17), "Pos LS: %i", text variable: UnitTesting.Sft_LS_PosLS
        OnMouseClick: write the text variable via Edit
    Rectangle (0,180 113x17), "Pos MS1: %i", text variable: UnitTesting.Sft_LS_PosMS1
        OnMouseClick: write the text variable via Edit
    Rectangle (0,200 113x17), "Pos MS2: %i", text variable: UnitTesting.Sft_LS_PosMS2
        OnMouseClick: write the text variable via Edit
    Frame (200,276 229x345)
        shows Vis_SafetyZone1(I_Title := 'SafetyZone 1', IO_SafetyLogic := MAIN.General.SafetyController)
    Button (12,24 61x21), "JogMin"
        tap UnitTesting.Sft_LS_JogBoxMin
    Button (88,24 61x21), "JogPlus"
        tap UnitTesting.Sft_LS_JogBoxPlus
    Rectangle (0,276 197x341)
    Button (8,416 181x21), "FB-K-ES", pressed state: UnitTesting.Sft_FB_K_ES_OK
        toggle UnitTesting.Sft_FB_K_ES_OK
    Button (8,440 181x21), "PS-Y1", pressed state: UnitTesting.Sft_Y_FB1
        toggle UnitTesting.Sft_Y_FB1
    Button (8,488 181x21), "PS-Y2", pressed state: UnitTesting.Sft_Y_FB2
        toggle UnitTesting.Sft_Y_FB2
    Button (8,368 57x21), "PB_ES", pressed state: UnitTesting.Sft_PB_ES
        toggle UnitTesting.Sft_PB_ES
    Button (8,320 181x21), "Enable = block simulation", pressed state: UnitTesting.Sft_EnableSafetyTest
        toggle UnitTesting.Sft_EnableSafetyTest
    Button (8,464 181x21), "PS-Y1 leaking", pressed state: UnitTesting.Sft_Y1_Leaking
        toggle UnitTesting.Sft_Y1_Leaking
    Button (8,512 181x21), "PS-Y2 leaking", pressed state: UnitTesting.Sft_Y2_Leaking
        toggle UnitTesting.Sft_Y2_Leaking
    Rectangle (0,276 197x45), "Unittesting >> Safety (requires special wiring)"
    Button (8,536 181x21), "Servo SLP ( -10 to + 10 pp)", pressed state: UnitTesting.Qsf_K_EnableSafePosition
        toggle UnitTesting.Qsf_K_EnableSafePosition
    Button (8,560 181x21), "Servo SLS (1000 incr/s)", pressed state: UnitTesting.Qsf_K_EnableSafeSpeed
        toggle UnitTesting.Qsf_K_EnableSafeSpeed
    Button (8,584 181x21), "Servo LS positive", pressed state: UnitTesting.LS_Positive.I_K_State
        toggle UnitTesting.LS_Positive.I_K_State
    Button (8,344 181x21), "Restart Safety"
        tap UnitTesting.Sft_PB_IllegalRestart
    Button (164,24 93x21), "Enable muting"
        toggle MAIN.General.SafetyController.I_K_EnableLsRejectMuting
    Rectangle (152,164 213x21), "State: %s", text variable: MAIN.General.SafetyController.LS_Entry1._HM_State
    Rectangle (364,164 25x21), "%i", text variable: MAIN.General.SafetyController.LS_Entry1._HM_State
    Ellipse (-8,72 20x20), colour toggle: MAIN.General.SafetyController.LS_Entry1.HMI.STS.StateMuted
        p3560616238: UnitTesting.Sft_LS_PosLS
    Rectangle (68,368 121x21), "State: %s", text variable: MAIN.General.SafetyController.PB_ES_MainCabinet._HM_State
    Button (8,392 181x21), "PB_ES_CHAN1 KAPUT"
        toggle UnitTesting.Sft_PB_ES_Chan1Broken
    Frame (432,276 142x262)
        shows BoikonLib.Vis_Organiser(I_UnitName := 'Organiser'', IO_cntrl_Organiser := MAIN.Organiser)
END_VISUALIZATION

// ---- General/Vis_General.TcVIS
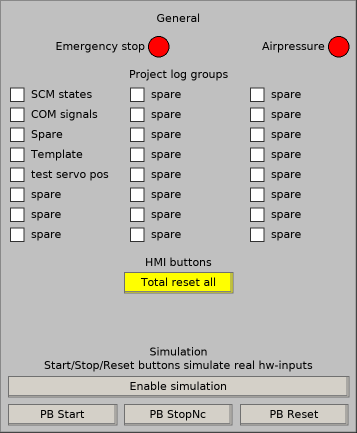
VISUALIZATION Vis_General  // 357x433
VAR_IN_OUT
	IO_General: utl_General;
END_VAR
    Rectangle (0,0 357x433)
    Rectangle (8,8 341x21), "General"
    Button (8,376 341x21), "Enable simulation"
        toggle Glbl.SimEnable
    Button (124,272 109x21), "Total reset all", pressed state: IO_General.PbSf_TotalResetAll.P_BypassStateTrue
        tap IO_General.PbSf_TotalResetAll.P_BypassStateTrue
    Checkbox (8,84 21x21), variable: BknLog.ActiveGroups.8
    Checkbox (8,104 21x21), variable: BknLog.ActiveGroups.9
    Checkbox (8,124 21x21), variable: BknLog.ActiveGroups.10
    Checkbox (8,164 21x21), variable: BknLog.ActiveGroups.12
    Checkbox (8,184 21x21), variable: BknLog.ActiveGroups.13
    Checkbox (8,204 21x21), variable: BknLog.ActiveGroups.14
    Checkbox (8,144 21x21), variable: BknLog.ActiveGroups.11
    Checkbox (8,224 21x21), variable: BknLog.ActiveGroups.15
    Label (28,84 81x21), "SCM states"
    Label (8,64 341x21), "Project log groups"
    Label (28,104 81x21), "COM signals"
    Label (28,124 81x21), "Spare"
    Label (28,144 81x21), "Template"
    Label (28,164 81x21), "test servo pos"
    Label (28,184 81x21), "spare"
    Label (28,204 81x21), "spare"
    Label (28,224 81x21), "spare"
    Checkbox (128,204 21x21), variable: BknLog.ActiveGroups.22
    Checkbox (128,224 21x21), variable: BknLog.ActiveGroups.23
    Checkbox (248,84 21x21), variable: BknLog.ActiveGroups.24
    Checkbox (128,184 21x21), variable: BknLog.ActiveGroups.21
    Checkbox (248,104 21x21), variable: BknLog.ActiveGroups.25
    Label (148,184 81x21), "spare"
    Label (148,204 81x21), "spare"
    Label (148,224 81x21), "spare"
    Label (268,84 81x21), "spare"
    Label (268,104 81x21), "spare"
    Checkbox (128,124 21x21), variable: BknLog.ActiveGroups.18
    Checkbox (128,144 21x21), variable: BknLog.ActiveGroups.19
    Checkbox (128,164 21x21), variable: BknLog.ActiveGroups.20
    Label (148,124 81x21), "spare"
    Label (148,144 81x21), "spare"
    Label (148,164 81x21), "spare"
    Checkbox (128,84 21x21), variable: BknLog.ActiveGroups.16
    Checkbox (128,104 21x21), variable: BknLog.ActiveGroups.17
    Label (148,84 81x21), "spare"
    Label (148,104 81x21), "spare"
    Checkbox (248,124 21x21), variable: BknLog.ActiveGroups.26
    Checkbox (248,144 21x21), variable: BknLog.ActiveGroups.27
    Label (268,124 81x21), "spare"
    Label (268,144 81x21), "spare"
    Checkbox (248,164 21x21), variable: BknLog.ActiveGroups.28
    Checkbox (248,184 21x21), variable: BknLog.ActiveGroups.29
    Label (268,164 81x21), "spare"
    Label (268,184 81x21), "spare"
    Checkbox (248,204 21x21), variable: BknLog.ActiveGroups.30
    Checkbox (248,224 21x21), variable: BknLog.ActiveGroups.31
    Label (268,204 81x21), "spare"
    Label (268,224 81x21), "spare"
    Rectangle (8,340 341x37), "Simulation Start/Stop/Reset buttons simulate real hw-inputs"
    Button (8,404 109x21), "PB Start"
        tap MAIN.General.I_Pb_StartAll.I_K_SimulateOn
    Button (124,404 108x21), "PB StopNc"
        toggle MAIN.General.I_PbNc_StopAll.I_K_SimulateOn
    Button (240,404 108x21), "PB Reset"
        tap MAIN.General.I_Pb_ResetAll.I_K_SimulateOn
    Label (8,252 341x21), "HMI buttons"
    Ellipse (148,36 21x21), colour toggle: IO_General.Q_SN_ES_Zone1_OK
    Label (0,36 148x21), "Emergency stop"
    Label (180,36 148x21), "Airpressure"
    Ellipse (328,36 21x21), colour toggle: MAIN.General.I_PS_AirpressureOk.HMI.STS.State
END_VISUALIZATION

// ---- GlobalTextList.TcGTLO
TEXTLIST GlobalTextList
  3440 = '\n\nHMI Buttons'
  1072 = '\nHMI Buttons'
  3494 = '\nHMI Buttons\n'
  183 = '\nHMI Buttons\na'
  719 = '\n15  14  13  12  11  10  09  08  00'
  341 = ' Machinename: %s'
  17 = '%2.1f KB/s'
  696 = '%f'
  98 = '%i'
  758 = '%I'
  18 = '%r KB/s'
  839 = '%s'
  1853 = '%s - state safety'
  264 = '%u'
  1387 = '%x'
  2138 = '(a general HMI-PB- start/stop/reset not implemented in the template, if you need it, go ahead)'
  3458 = '(pb start/stop/reset not implemented in the template, if you need it, go ahead)'
  818 = '10: %s'
  682 = '15  14  13  12  11  10  09  08'
  485 = '15  14  13  12  11  10  09  08  00'
  273 = '1: %s'
  724 = '2: %s'
  892 = '3: %s'
  234 = '4: %s'
  635 = '5: %s'
  589 = '6: %s'
  412 = '7: %s'
  26 = '8: %s'
  299 = '9: %s'
  1228 = '<<'
  42 = '<<<'
  179 = '>-1 then used for autocal'
  142 = '>>'
  1054 = '@Error 6 >> Install/Repair the TCP-IP option'
  2481 = 'a'
  67 = 'Activate ext sp mode'
  263 = 'Activate simulation'
  702 = 'Activate stepmodus'
  463 = 'Active logging groups \n(eLogGroups defines bits)'
  649 = 'Active logging groups \n07    06  05  04  03  02  01  00'
  669 = 'Active logging groups \n07  06  05  04  03  02  01  00'
  816 = 'Active logging groups \n07 06  05  04  03  02  01  00'
  25 = 'Active logging groups \n15  14  13  12  11  10  09  08  07  06  05  04  03  02  01  00'
  168 = 'Active logging groups \n15 14 13 12 11 10 09 08 07 06 05 04 03 02 01 00'
  47 = 'Active recipe per group'
  317 = 'Active recipes per group'
  1591 = 'Active scene/group: %s'
  1547 = 'Address: %i'
  558 = 'Airpressure'
  2393 = 'All Ok'
  86 = 'Analogs'
  507 = 'ApptimeStamp: %s'
  323 = 'At speed'
  821 = 'Auto ExtSpMode'
  636 = 'Auto Velo: %.2f'
  12 = 'Auto Velo: %2.2f'
  1630 = 'AutoCal'
  292 = 'Base position: %i'
  2791 = 'Batt life: %i %%'
  3556 = 'Batt life: %s'
  2624 = 'Battery life: %i %%'
  660 = 'buffer max level: %i %%'
  1306 = 'buffer overflows: %i'
  94 = 'Calc claws open dst: %.1f'
  1725 = 'Calculated claws dst: %.1f'
  258 = 'Calculated claws dst: %f.1'
  1336 = 'Call Houston'
  1396 = 'Cmnd rcv: %i ms'
  993 = 'Cmnd send: %i ms'
  909 = 'Cmnd(ms): %i'
  1266 = 'cntr err'
  527 = 'Cntrl'
  956 = 'cntrl states'
  250 = 'COM signals'
  685 = 'Config'
  396 = 'Config: %s'
  4469 = 'Confirm Dumped'
  3258 = 'Confirm Empty'
  49 = 'Confirm Payload'
  369 = 'Cpu load: %2.1f'
  743 = 'Cpu load: %2.1f %%'
  1035 = 'CRC: %h'
  2050 = 'CRC: %x'
  3163 = 'CRC: 0x%x'
  632 = 'Current %s'
  469 = 'Current %u'
  38 = 'Current: %d'
  623 = 'Current: %s'
  3735 = 'Current: %s%'
  1160 = 'CurrentLimit'
  1404 = 'Cycle exec time: %2.2f ms'
  1827 = 'Danger!!!\nOnly for boikon engineers'
  1697 = 'Danger!!! /nOnly for boikon engineer'
  805 = 'Danger!!! Only for boikon engineer'
  693 = 'Debug Auto_ExtSpGen'
  2589 = 'Debug block inputs REMOVE ME'
  728 = 'Debug I_K_Auto_ExtSpmode'
  229 = 'Debug I_K_Auto_Velocity'
  274 = 'Debug I_K_ExtSpmode'
  868 = 'Debug Template State: %s'
  421 = 'Debug Velocity tets'
  608 = 'Default'
  424 = 'Diag: %i'
  3729 = 'Disable Block'
  498 = 'Disable LS'
  1624 = 'dr err'
  3156 = 'DR ES'
  1349 = 'DR ES (NC)'
  190 = 'Drive error bit'
  7 = 'Drive: %s'
  1618 = 'drv err'
  289 = 'DRV: %s'
  272 = 'Emergency stop'
  677 = 'Enable'
  3109 = 'Enable = block simulation'
  555 = 'Enable Array Tests'
  1448 = 'Enable camera'
  2077 = 'Enable I safety inputs sim'
  4767 = 'Enable muting'
  253 = 'Enable Run'
  4201 = 'Enable simulation'
  3397 = 'Enable Timer tests'
  566 = 'EnableStepLock'
  1546 = 'err'
  1440 = 'Err'
  1284 = 'Err ID textdisplay: %i'
  235 = 'Err ID: %i'
  1211 = 'Err: %s'
  1423 = 'ErrNr: %i'
  96 = 'Error'
  1496 = 'Error change cnt: %s'
  390 = 'Error changes: %s'
  1128 = 'Error ID   @Error 6 >> Install/Repair the TCP-IP option'
  108 = 'Error ID: %i'
  2426 = 'Error: %i'
  3557 = 'Error: %x'
  61 = 'ErrorNr: %I'
  2887 = 'ErrorNr: %i'
  1491 = 'ErrorNr: %x'
  3051 = 'ErrorNr:#16 %x'
  1912 = 'errors'
  1467 = 'Errors'
  832 = 'ES Air Active'
  2528 = 'ES Air ok'
  53 = 'ES Ok'
  2919 = 'ES Zone Ok'
  382 = 'ES Zone Ok TOF'
  2042 = 'ES Zone1'
  236 = 'ES Zone1 Ok'
  4777 = 'ES Zone2'
  148 = 'ES Zone2 Ok'
  1003 = 'ES ZoneAll'
  990 = 'ES_Air ok'
  244 = 'ES_ZoneOk'
  1527 = 'ES_ZoneOk_TOF'
  24 = 'Ethercatmanager %s'
  1702 = 'exp:%i'
  2904 = 'FB-K-ES'
  4337 = 'FB-Y1'
  1615 = 'FB-Y2'
  953 = 'FB_OK'
  490 = 'Feedback'
  1082 = 'focus:%i'
  2939 = 'ForceResultOk'
  153 = 'Fwd'
  1001 = 'gain:%i'
  254 = 'General'
  1283 = 'Get group/scene'
  2002 = 'Get status'
  814 = 'Grip Force: %i'
  3669 = 'GROTE TESTKNOP'
  959 = 'Group%i'
  588 = 'Group:%i'
  159 = 'HMI alive check tag: %s'
  2914 = 'HMI buttons'
  1534 = 'HMI Reset all organisers via\nGeneral.Q_SN_TotalReset'
  3252 = 'HMI Reset all organisers via\nHMI Buttons'
  1524 = 'Home'
  893 = 'Homed'
  87 = 'Homing mode: %i'
  1233 = 'HW-Trig'
  1308 = 'ID: %s'
  920 = 'if >-1 then autocal will use this value'
  2858 = 'Illegal safety restart button'
  937 = 'In'
  2455 = 'In Error'
  2198 = 'In Run'
  2948 = 'InError'
  410 = 'Info per slave'
  2699 = 'Info selected slave'
  1107 = 'Info selected slave index'
  1167 = 'Init left'
  459 = 'Init Right'
  114 = 'Inputs'
  447 = 'IP address: %s'
  195 = 'IP port: %s'
  1227 = 'ip:%s'
  3514 = 'I_K_SelectProg'
  1857 = 'Job: %s'
  1093 = 'Jog'
  337 = 'Jog +'
  665 = 'Jog -'
  1566 = 'Jog IS'
  452 = 'Jog OS'
  788 = 'Jog Speed: %2.2f'
  1817 = 'JogMin'
  2977 = 'JogPlus'
  206 = 'Last Cmnd: %s'
  2279 = 'Last command (ms): %i'
  100 = 'Last cycle time: %2.1f'
  952 = 'Last cycle time: %2.1f ms'
  691 = 'Last cycle time: %2.2f ms'
  9 = 'Last cycle time: %2.3f ms'
  2877 = 'Last trigger (ms):'
  1683 = 'Last trigger (ms): %i'
  170 = 'Library log groups'
  51 = 'Load Scene'
  2056 = 'LoadJob'
  1435 = 'LoadScene'
  585 = 'Logger alive'
  60 = 'Logger buffer max fill level: %i'
  736 = 'Logger buffer max fill level: %i %%'
  958 = 'Logger buffer min fill level: %i'
  445 = 'Logger buffer min fill level: %i %%'
  52 = 'Logger connected'
  401 = 'Logger log all channels'
  339 = 'Logger logging to file'
  356 = 'Logger machine name: %s'
  996 = 'Logger out of\nbool channels'
  986 = 'Logger out of\ndint channels'
  626 = 'Logger out of\nreal channels'
  535 = 'Logger paused'
  2544 = 'LS ES'
  1345 = 'LS ES (NC)'
  362 = 'M-Switch'
  807 = 'MAIN.HMI_Setpoints.TestingArea.PositionOffsetMatrix.PosOffsMatrix[0,0]._R'
  308 = 'MAIN.HMI_Setpoints.TestingArea.PositionOffsetMatrix.PosOffsMatrix[0,INDEX]._R'
  1925 = 'Manuals:'
  326 = 'Max cpu load: %2.1f'
  885 = 'Max cpu load: %2.1f %%'
  457 = 'Max cycle time: %2.1f'
  2 = 'Max cycle time: %2.1f ms'
  946 = 'Max cycle time: %2.2f ms'
  1444 = 'Max exec time: %2.2f ms'
  4802 = 'mijn voorbeeld %s'
  297 = 'Move Mode'
  841 = 'Move mode: %i'
  1447 = 'Move mode: %s'
  1199 = 'MQTT'
  670 = 'MQTT logger Setpoints'
  2359 = 'MQTT logging'
  822 = 'MQTT Setpoints'
  386 = 'MQTT-client state'
  57 = 'MS1'
  3322 = 'MS2'
  523 = 'MS_OK'
  4890 = 'Muted'
  2142 = 'Muting active'
  2272 = 'Name: %s'
  377 = 'Next'
  966 = 'Next NOP'
  1249 = 'NOTE: \nThe library groups are defined in the library\nThe project groups can be changed as needed'
  1400 = 'NOTE: \nThe library groups fixed\nThe project groups can be changed as needed'
  571 = 'NOTE: \nThe library groups should not be altered\nThe project groups can be changed as needed'
  1007 = 'NOTE: \nThe library groups should not be changed\nThe project groups can be changed as needed'
  501 = 'NOTE: adapt project logger groups\nas needed'
  321 = 'NOTE: adapt project logger groups as needed'
  941 = 'Nr NOP slaves: %i'
  1234 = 'Nr of found configured slaves'
  204 = 'Nr slaves: %i'
  4498 = 'Nr: %i '
  605 = 'NrPicks: %i'
  985 = 'Number of changes detected in HMI_Errors  (if count increases, then the HMI will update errors)'
  923 = 'Number of changes detected in the errors (if count increases, then the HMI will update errors)'
  1888 = 'Number of changes detected in the HMI_Warnings (if count increases, then the HMI will update errors)'
  2008 = 'Online change cnt: %s'
  785 = 'Online change count: %s'
  197 = 'Online changes: %s'
  1346 = 'Only for boikon engineer'
  2357 = 'Only to be used by boikon programmers'
  663 = 'Out'
  1562 = 'Output enabled'
  3341 = 'Output state'
  1716 = 'Output: %s'
  255 = 'Outputs'
  1085 = 'Overwrite HW-input buttons (only works if not linked)'
  2407 = 'Part result'
  91 = 'PayloadNr: %i'
  1212 = 'PB ES MCC'
  241 = 'PB ES MCC (NO)'
  537 = 'PB Reset'
  1783 = 'PB SafetyErrorReset'
  3780 = 'PB Start'
  2442 = 'PB Stop'
  1442 = 'PB StopNc'
  1880 = 'PB_ES'
  2498 = 'PB_ES_CHAN1 KAPUT'
  1969 = 'Pers. save failed'
  1874 = 'Persistent save cnt: %s'
  1603 = 'Persistent saves: %s'
  3381 = 'plc block in error'
  978 = 'PLC cycle time high'
  852 = 'Plcblock State: %s'
  1646 = 'port:%i'
  1847 = 'Pos LS: %I'
  2270 = 'Pos LS: %i'
  3813 = 'Pos MS1: %i'
  3111 = 'Pos MS2: %i'
  1693 = 'Pos tolerance: %i'
  425 = 'Position: %u'
  336 = 'Prev'
  2015 = 'Prev NOP'
  2680 = 'Project dependant statusses'
  32 = 'Project log groups'
  884 = 'Project name: %s'
  2839 = 'PS-Y1'
  3242 = 'PS-Y1 ForceOff'
  2938 = 'PS-Y1 leaking'
  4034 = 'PS-Y2'
  1330 = 'PS-Y2 ForceOff'
  1193 = 'PS-Y2 leaking'
  828 = 'QuickFocus'
  101 = 'R'
  1777 = 'Raw result: %s'
  2622 = 'RBT: %s'
  1766 = 'Rcv Msg: %s'
  1147 = 'Read group/scene'
  1476 = 'Read group/state'
  858 = 'Ready'
  75 = 'ref ok'
  1310 = 'Rescan'
  411 = 'Reset'
  59 = 'Reset all organisers via\nGeneral.Q_SN_TotalReset'
  483 = 'Reset all organisers via\nGeneral.Q_SN_TotalReset\n'
  914 = 'Reset all organisers via General.Q_SN_TotalReset\n'
  2340 = 'Reset program error'
  520 = 'Reset Safety Logic Error'
  1695 = 'Response: %i ms'
  1850 = 'RESTART ONLY FOR UNITTESTING'
  967 = 'Restart safety'
  4488 = 'Restart Safety'
  198 = 'Restart safety DANGER'
  2421 = 'Restart slave'
  2060 = 'Restart this slave'
  239 = 'Result: %s'
  208 = 'Results:'
  270 = 'Rev'
  1608 = 'Robot signals (normally auto controlled)'
  1384 = 'Run'
  220 = 'Running'
  213 = 'Runtime: %s h'
  128 = 'Runtime: %s s'
  622 = 'Runtime: %u'
  536 = 'S: %s'
  863 = 'Safety Enable SIM'
  68 = 'Safety In run'
  181 = 'Safety SIM FB K ES'
  2707 = 'Safety SIM FB Y PS1'
  1641 = 'Safety SIM FB Y PS2'
  1563 = 'Safety SIM PB ES'
  1664 = 'Safety SIM Y1 Leaking'
  573 = 'Safety zone 1 OK'
  1722 = 'Safety: sim inputs real safety cards with plc output cards'
  1210 = 'Safety: sim inputs sf cards\n with plc output cards'
  1482 = 'Safety: sim inputs sf cards\n with plc output cards.\nNeeds to be wired in correct way'
  602 = 'Saving setpoints failed'
  3299 = 'Scene:%i'
  290 = 'SceneNr: %s'
  182 = 'SCM states'
  637 = 'SCM_TemplateMachinePart State: %s'
  835 = 'Send Cmnd: %s'
  1127 = 'Sero LS positive'
  780 = 'Service >> first check and fix reason of error'
  2718 = 'Servo LS positive'
  4447 = 'Servo SLP'
  318 = 'Servo SLP ( -10 to + 10 pp)'
  2466 = 'Servo SLP (safe pos -10 to + 10 polepairs'
  102 = 'Servo SLS'
  4487 = 'Servo SLS (1000 incr/s)'
  4069 = 'Servo SLS (1000incr/s)'
  3410 = 'Servo SLS (safe speed)'
  731 = 'Set cycle time: %.1f'
  656 = 'Set cycle time: %.1f ms'
  606 = 'Set cycle time: %2.1f'
  1064 = 'Set Group'
  259 = 'Set master state'
  981 = 'Set Scene'
  44 = 'Setpoint: Logger machine name: %s'
  824 = 'Setpoints'
  1287 = 'Setpoints:'
  385 = 'SFT-group HW: %s'
  1417 = 'SFT-group Z-ALL: %s'
  5074 = 'SFT-group Z2: %s'
  4685 = 'SFT-group zone 1: %s'
  3502 = 'SFT-groupZ1: %s'
  480 = 'Shift position: %i'
  1686 = 'Show slave state info selected index: %i'
  830 = 'Show state info selected index: %i'
  1 = 'sim i safety fb k es'
  1887 = 'sim i safety fb y1'
  203 = 'sim i safety fb y2'
  2505 = 'sim i safety pb es'
  173 = 'Sim myMachinePart'
  512 = 'Sim PB Reset'
  192 = 'Sim PB Start'
  628 = 'Sim PB Stop'
  655 = 'Sim PB TotalReset'
  306 = 'Sim TemplateMachinePart'
  895 = 'Simulate emergencystop circuit OK'
  2689 = 'Simulate general start/stop/reset buttons'
  1617 = 'Simulation'
  90 = 'Simulation\nStart/Stop/Reset buttons simulate real hw-inputs'
  1875 = 'Simulation >> sim hw-buttons'
  1111 = 'Simulation >>will simulate the hardware buttons'
  2102 = 'Slave Index: %2.2f% '
  15 = 'Slave Index: %i'
  1764 = 'Slaves not in "OP" state'
  746 = 'SP save to disk count: %s'
  992 = 'spare'
  1449 = 'Spare'
  508 = 'Speed: %2.2f% '
  1258 = 'Speed: %d '
  700 = 'Speed: %i% '
  957 = 'Speed: %s'
  423 = 'Speed: %s%'
  0 = 'Speed: %u'
  591 = 'Start'
  2233 = 'state %s'
  1422 = 'State: %i'
  1267 = 'State: %i %s'
  820 = 'State: %s'
  831 = 'state: %s'
  745 = 'State: 0x %s'
  1775 = 'State: 0x%s'
  1356 = 'Statusses'
  3743 = 'Statusses from twinsafe'
  1497 = 'Statusses plc inputs'
  2866 = 'Stop'
  924 = 'Strokes: %s'
  3929 = 'STS in error'
  639 = 'Sts: %s'
  66 = 'switch'
  521 = 'TargetPos: %2.2f'
  311 = 'Teach position: %i'
  878 = 'template'
  968 = 'Template'
  714 = 'test servo pos'
  3346 = 'testBool'
  800 = 'testing area'
  3858 = 'testInt: %i'
  3384 = 'testInt: %s'
  2385 = 'testReal: %f'
  3329 = 'testReal: %i'
  1097 = 'Time Cmnd %i'
  1954 = 'Time Cmnd%i'
  2995 = 'Time Cmnd: %i'
  1799 = 'Time Trigger %i'
  811 = 'Time Trigger: %i'
  2712 = 'Time: %i ms'
  489 = 'Time: %s'
  1033 = 'TimeCmnd: %i ms'
  1118 = 'timeout:%i ms'
  1612 = 'timeout:%s'
  1241 = 'TimeSend: %i ms'
  562 = 'To Base'
  629 = 'To Work'
  1299 = 'Toggle group'
  1341 = 'Toggle Run/Stop'
  486 = 'ToggleExtSpMode'
  5 = 'Total reset all'
  2990 = 'Trig timeout%i'
  1291 = 'Trig timeout: %d'
  2071 = 'Trig timeout: %i'
  1337 = 'Trig timeout: %s'
  1275 = 'Trig timeout: %t'
  1483 = 'Trig timeout:%i'
  567 = 'Trigger'
  2943 = 'Trigger(ms)'
  2378 = 'Trigger(ms):'
  1604 = 'Twinsafe control'
  28 = 'UNIT TEST FAILED'
  1962 = 'UnitTest > EnablePosDir'
  215 = 'UnitTest Enable'
  2095 = 'UnitTest Enable sf inputs'
  651 = 'UnitTest FB-k-ES'
  3067 = 'UnitTest FB-K-ES'
  4374 = 'UnitTest FB-Y1'
  1828 = 'UnitTest FB-Y2'
  2931 = 'UnitTest PbEs'
  664 = 'UnitTest PB_ES'
  2384 = 'UnitTesting'
  960 = 'UnitTesting (only for library debugging)'
  1076 = 'Unittesting >> Safety \n(requires special wiring)'
  683 = 'Unittesting >> Safety (requires special wiring)'
  1295 = 'UnlockStep'
  172 = 'UPS batterymode'
  3883 = 'Ups Error'
  2499 = 'Ups on battery'
  340 = 'Ups warning active'
  998 = 'Ups warning: %s'
  127 = 'Use HW-trigger'
  11 = 'Velocity: %i'
  3374 = 'Version: %s'
  1034 = 'Warning actual config paras!'
  630 = 'Warning change cnt: %s'
  1074 = 'Warning changes: %s'
  979 = 'Work position: %i'
  358 = 'X'
  1209 = 'X:%i'
  420 = 'Y'
  1002 = 'Y1 is leaking'
  3053 = 'Y2 is leaking'
  1429 = 'Y:%i'
  2907 = 'Zone1 OK'
  3345 = 'Zone2 OK'
  1899 = 'Zones'
END_TEXTLIST

// ---- Main/VisGeneral.TcVIS
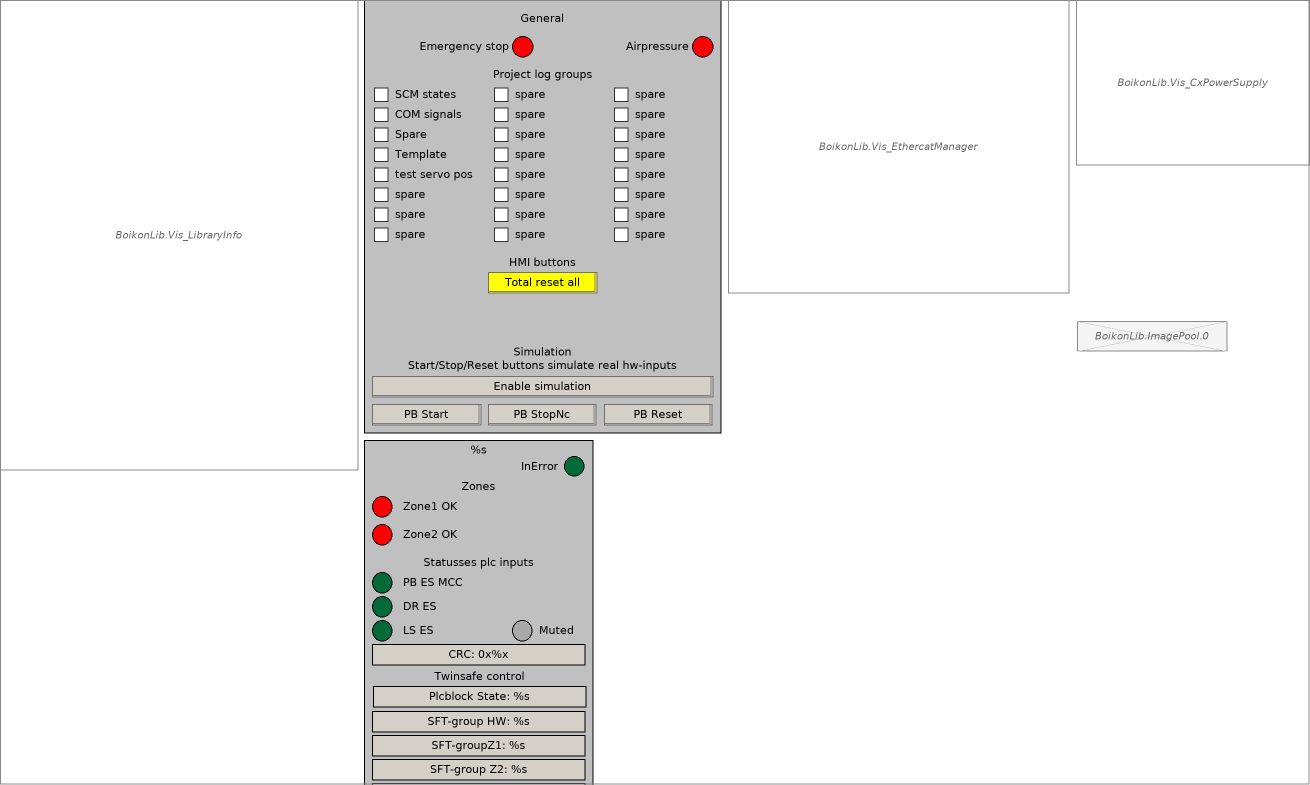
VISUALIZATION VisGeneral  // 1310x785, background image BoikonLib.Images.0
    Frame (364,0 361x437)
        shows Vis_General(IO_General := MAIN.General)
    Frame (728,0 341x293)
        shows BoikonLib.Vis_EthercatManager(IO_EM := MAIN.General.EthercatManager)
    Frame (364,440 229x345)
        shows Vis_SafetyZone1(I_Title := 'SafetyZone 1', IO_SafetyLogic := MAIN.General.SafetyController)
    Frame (1076,0 234x165)
        shows BoikonLib.Vis_CxPowerSupply(I_Title := 'cx power supply', IO := MAIN.General.CxPowerSupply)
    Frame (0,0 358x470)
        shows BoikonLib.Vis_LibraryInfo(IO_Cntrl := MAIN.General.BknLibrary)
    Image (569,383 0x1), image: BoikonLib.ImagePool.0
    Image (1077,321 150x30), image: BoikonLib.ImagePool.0
END_VISUALIZATION

// ---- Main/VisScmTemplate.TcVIS
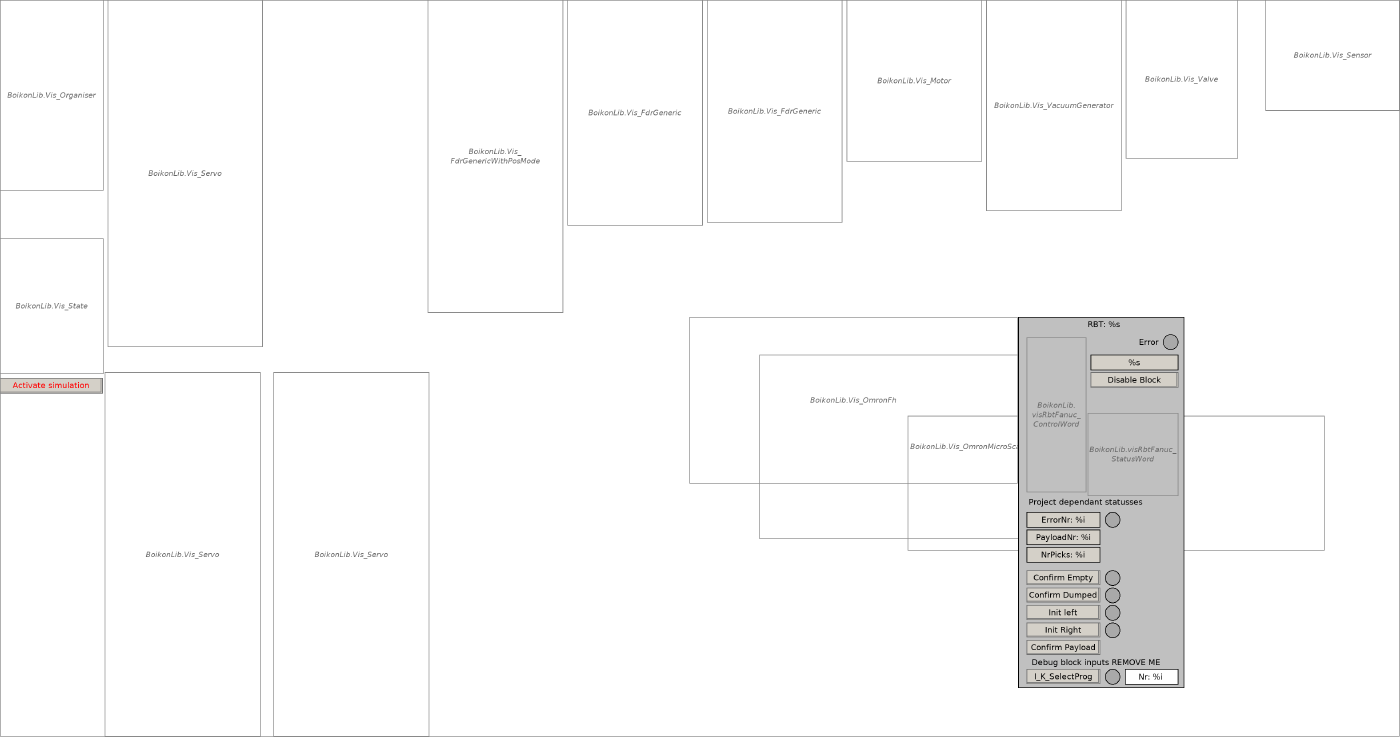
VISUALIZATION VisScmTemplate  // 1925x1014
    Frame (148,0 213x477)
        shows BoikonLib.Vis_Servo(I_UnitName := 'Xaxis', IO_cntrl_Servo := MAIN.ExampleMachinePart.Srv_Xaxis)
    Button (0,520 141x21), "Activate simulation"
        toggle Glbl.Sim_MyMachinePart
    Frame (1044,488 573x253)
        shows BoikonLib.Vis_OmronMicroScan(I_UnitName := 'Omron Smart Cam', IO_cntrl := MAIN.ExampleMachinePart.Cam_OmronSmartCam)
    Frame (948,436 451x229)
        shows BoikonLib.Vis_OmronFh(I_UnitName := 'OmronFh', IO_cntrl := MAIN.ExampleMachinePart.Cam_OmronFh)
    Frame (1740,0 185x152)
        shows BoikonLib.Vis_Sensor(I_UnitName := 'Example sensor', IO_cntrl := MAIN.ExampleMachinePart.PC_ProductInfeed)
    Frame (1548,0 154x218)
        shows BoikonLib.Vis_Valve(I_UnitName := 'TempValve', IO_cntrl := MAIN.ExampleMachinePart.Cyl_Example)
    Frame (1356,0 186x290)
        shows BoikonLib.Vis_VacuumGenerator(I_UnitName := 'VacuumGenerator', IO := MAIN.ExampleMachinePart.Vcg_Suckers)
    Frame (1248,572 573x185)
        shows BoikonLib.Vis_OmronFhEth(I_UnitName := 'OmronEth', IO_cntrl := MAIN.ExampleMachinePart.Cam_OmronFhEth)
    Frame (972,0 186x306)
        shows BoikonLib.Vis_FdrGeneric(I_UnitName := 'Lenze', IO_Cntrl := MAIN.ExampleMachinePart.Fdr_LzExample)
    Frame (780,0 186x310)
        shows BoikonLib.Vis_FdrGeneric(I_UnitName := 'ControlTech', IO_Cntrl := MAIN.ExampleMachinePart.Fdr_CtExample)
    Frame (1164,0 186x222)
        shows BoikonLib.Vis_Motor(I_UnitName := 'Example', IO_cntrl := MAIN.ExampleMachinePart.Mtr_Example)
    Frame (0,0 142x262)
        shows BoikonLib.Vis_Organiser(I_UnitName := 'Organiser'', IO_cntrl_Organiser := MAIN.Organiser)
    Frame (588,0 186x430)
        shows BoikonLib.Vis_FdrGenericWithPosMode(I_UnitName := 'Interrol', IO_Cntrl := MAIN.ExampleMachinePart.Srv_Interrol)
    Frame (0,328 142x186)
        shows BoikonLib.Vis_State(I_UnitName := 'SCM state', IO_Step := MAIN.ExampleMachinePart.State)
    Frame (1400,436 248x510)
        shows Vis_RbtFanucUnloading(I_UnitName := 'Unloading', IO_cntrl := MAIN.ExampleMachinePart.Rbt_Unloading)
    Frame (144,512 214x502)
        shows BoikonLib.Vis_Servo(I_UnitName := 'Yaxis', IO_cntrl_Servo := MAIN.ExampleMachinePart.Srv_Yaxis)
    Frame (376,512 214x502)
        shows BoikonLib.Vis_Servo(I_UnitName := 'Zaxis', IO_cntrl_Servo := MAIN.ExampleMachinePart.Srv_Zaxis)
END_VISUALIZATION

// ---- _Control_Templates/cntrl_RbtFanuc/HMI/Vis_RbtFanucUnloading.TcVIS
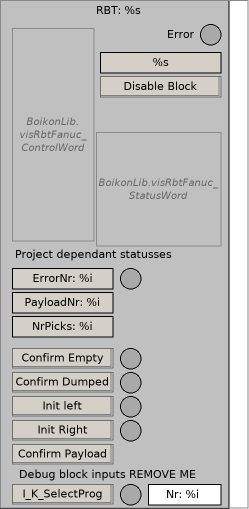
VISUALIZATION Vis_RbtFanucUnloading  // 249x509
VAR_INPUT
	I_UnitName:STRING := 'myRobot';
END_VAR

VAR_IN_OUT
	IO_cntrl: cntrl_RbtFanucUnloadingRobot;
END_VAR
    Rectangle (0,0 229x509)
    Rectangle (4,0 229x21), "RBT: %s", text variable: I_UnitName
    Frame (12,28 82x213)
        shows BoikonLib.visRbtFanuc_ControlWord(IO := IO_cntrl.Q_DataOut.Vars._UI)
    Frame (96,132 125x114)
        shows BoikonLib.visRbtFanuc_StatusWord(IO := IO_cntrl.I_DataIn.Vars._UO)
    Button (100,76 121x21), "Disable Block"
        toggle IO_cntrl.TB_DisableActivations
    Ellipse (120,348 21x21), colour toggle: IO_cntrl.I_DataIn.Vars._DO.SN_CrateEmpty
    Button (12,348 101x20), "Confirm Empty"
        tap IO_cntrl.Q_DataOut.Vars._DI.SN_CrateEmptyOk
    Rectangle (12,316 101x21), "NrPicks: %i", text variable: IO_cntrl.I_DataIn.Vars._GO.NrPickedCrates
    Button (12,372 101x20), "Confirm Dumped"
        tap IO_cntrl.Q_DataOut.Vars._DI.SN_RequestDumpOk
    Ellipse (120,372 21x21), colour toggle: IO_cntrl.I_DataIn.Vars._DO.SN_RequestDump
    Ellipse (120,396 21x21), colour toggle: IO_cntrl.I_DataIn.Vars._DO.SN_InitLeftOk
    Ellipse (120,420 21x21), colour toggle: IO_cntrl.I_DataIn.Vars._DO.SN_InitRightOk
    Button (12,396 101x20), "Init left"
        toggle IO_cntrl.Q_DataOut.Vars._DI.SN_InitLeft
    Button (12,420 101x20), "Init Right"
        toggle IO_cntrl.Q_DataOut.Vars._DI.SN_InitRight
    Ellipse (120,268 21x21), colour toggle: IO_cntrl.I_DataIn.Vars._DO.STS_Error
    Rectangle (12,268 101x21), "ErrorNr: %i", text variable: IO_cntrl.I_DataIn.Vars._GO.ErrorNr
    Button (12,444 101x20), "Confirm Payload"
        tap IO_cntrl.Q_DataOut.Vars._DI.SN_PayloadConfirm
    Rectangle (12,292 101x21), "PayloadNr: %i", text variable: IO_cntrl.I_DataIn.Vars._GO.NrPayload
    Label (12,248 209x13), "Project dependant statusses"
    Label (16,468 233x13), "Debug block inputs REMOVE ME"
    Button (12,484 101x20), "I_K_SelectProg"
        toggle IO_cntrl.I_K_ProgramSelect
    Ellipse (120,484 21x21), colour toggle: IO_cntrl.Q_K_ProgramSelect_OK
    Rectangle (148,484 73x21), "Nr: %i", text variable: IO_cntrl.I_SP_ProgramNr
        OnMouseClick: write the text variable via Default, min 0, max 100
    Rectangle (100,52 121x21), "%s", text variable: IO_cntrl.eS
    Label (148,24 49x21), "Error"
    Ellipse (200,24 21x21), colour toggle: IO_cntrl.HMI.P_STS_InError
END_VISUALIZATION

// ---- _Control_Templates/cntrl_SafetyController/Vis_SafetyZone1.TcVIS
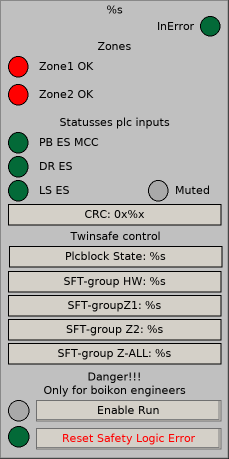
VISUALIZATION Vis_SafetyZone1  // 229x459
VAR_INPUT
	I_Title:string;
END_VAR

VAR_IN_OUT
	IO_SafetyLogic:cntrl_SafetyController1;
END_VAR
    Rectangle (0,0 229x459)
    Rectangle (12,0 205x20), "%s", text variable: I_Title
    Rectangle (9,246 213x21), "Plcblock State: %s", text variable: IO_SafetyLogic.eS
    Button (36,428 185x21), "Reset Safety Logic Error", pressed state: IO_SafetyLogic.PbSf_ResetSafetyErrors.P_BypassStateTrue
        tap IO_SafetyLogic.PbSf_ResetSafetyErrors.P_BypassStateTrue
    Ellipse (8,426 21x21), colour toggle: IO_SafetyLogic.HMI.STS.LogicInError
    Ellipse (8,400 21x21), colour toggle: IO_SafetyLogic.HMI.STS.LogicRunning
    Rectangle (8,368 213x31), "Danger!!! Only for boikon engineers"
    Button (36,400 185x21), "Enable Run", pressed state: IO_SafetyLogic.HMI.STS.PB_RunSafetyLogic
        toggle IO_SafetyLogic.HMI.STS.PB_RunSafetyLogic
    Ellipse (8,56 20x21), colour toggle: IO_SafetyLogic.SFG_Zone1_Run.HMI.STS.StateOk
    Rectangle (36,56 181x21), "Zone1 OK"
    Ellipse (8,132 20x21), colour toggle: NOT IO_SafetyLogic.PB_ES_MainCabinet.HMI.STS.StateOk
    Rectangle (36,132 181x21), "PB ES MCC"
    Ellipse (8,156 20x21), colour toggle: NOT IO_SafetyLogic.DR_Front.HMI.STS.StateOk
    Rectangle (36,156 181x21), "DR ES"
    Ellipse (8,180 20x21), colour toggle: NOT IO_SafetyLogic.LS_Entry1.HMI.STS.StateOk
    Rectangle (36,180 73x21), "LS ES"
    Ellipse (200,16 20x20), colour toggle: IO_SafetyLogic.HMI.P_STS_InError
    Rectangle (128,16 69x21), "InError"
    Label (8,36 213x21), "Zones"
    Label (8,112 213x21), "Statusses plc inputs"
    Label (9,226 213x21), "Twinsafe control"
    Rectangle (8,204 213x21), "CRC: 0x%x", text variable: IO_SafetyLogic.HMI.STS.CrcCodeProject
    Ellipse (8,84 20x21), colour toggle: IO_SafetyLogic.SFG_Zone2_Run.HMI.STS.StateOk
    Rectangle (36,84 181x21), "Zone2 OK"
    Ellipse (148,180 20x21), colour toggle: IO_SafetyLogic.LS_Entry1.HMI.STS.StateMuted
    Rectangle (172,180 49x21), "Muted"
    Rectangle (8,271 213x21), "SFT-group HW: %s", text variable: IO_SafetyLogic.SFG_Hardware_Run._HM_State
    Rectangle (8,295 213x21), "SFT-groupZ1: %s", text variable: IO_SafetyLogic.SFG_Zone1_Run._HM_State
    Rectangle (8,319 213x21), "SFT-group Z2: %s", text variable: IO_SafetyLogic.SFG_Zone2_Run._HM_State
    Rectangle (8,343 213x21), "SFT-group Z-ALL: %s", text variable: IO_SafetyLogic.SFG_ZoneAll_Run._HM_State
END_VISUALIZATION
